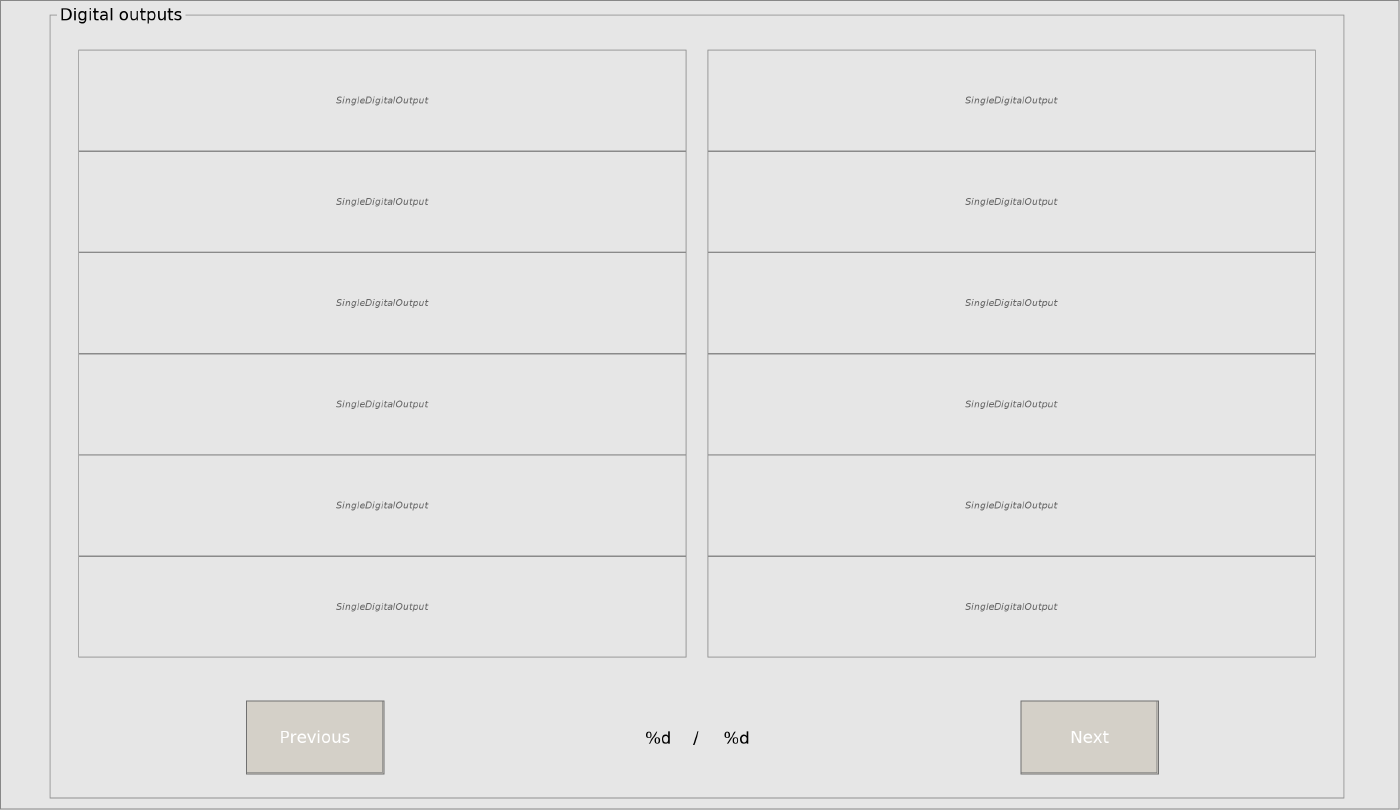
VISUALIZATION PageManualOutputs  // 1520x880
VAR_IN_OUT
	btnPrevious			: BOOL;
	btnNext				: BOOL;
	
	bPreviousInvisible	: BOOL;
	bNextInvisible		: BOOL;
	
	stDigitalOutputEmpty: ARRAY[1..12] OF BOOL;
	stDigitalOutputData	: ARRAY[1..12] OF ST_VisuCtrlOutputFrame;
	
	iOutputSelectedPageIndex	: USINT;
	iOutputTotalPageIndex 		: USINT;
END_VAR
    GroupBox (54,8 1405x859), "Digital outputs"
        Rectangle (721,769 50x50), "%d", text variable: iOutputTotalPageIndex + 1
        Rectangle (636,769 50x50), "%d", text variable: iOutputSelectedPageIndex+1
        Rectangle (636,768 131x51), "/"
        Button (213,753 150x80), "Previous", invisible if: bPreviousInvisible
            tap btnPrevious
        Button (1054,753 150x80), "Next", invisible if: bNextInvisible
            tap btnNext
        Frame (31,46 660x110), invisible if: stDigitalOutputEmpty[1]
            shows SingleDigitalOutput(stDigitalOutput := stDigitalOutputData[1])
        Frame (31,156 660x110), invisible if: stDigitalOutputEmpty[2]
            shows SingleDigitalOutput(stDigitalOutput := stDigitalOutputData[2])
        Frame (31,266 660x110), invisible if: stDigitalOutputEmpty[3]
            shows SingleDigitalOutput(stDigitalOutput := stDigitalOutputData[3])
        Frame (31,376 660x110), invisible if: stDigitalOutputEmpty[4]
            shows SingleDigitalOutput(stDigitalOutput := stDigitalOutputData[4])
        Frame (31,486 660x110), invisible if: stDigitalOutputEmpty[5]
            shows SingleDigitalOutput(stDigitalOutput := stDigitalOutputData[5])
        Frame (31,596 660x110), invisible if: stDigitalOutputEmpty[6]
            shows SingleDigitalOutput(stDigitalOutput := stDigitalOutputData[6])
        Frame (714,46 660x110), invisible if: stDigitalOutputEmpty[7]
            shows SingleDigitalOutput(stDigitalOutput := stDigitalOutputData[7])
    Frame (768,164 660x110), invisible if: stDigitalOutputEmpty[8]
        shows SingleDigitalOutput(stDigitalOutput := stDigitalOutputData[8])
    Frame (768,274 660x110), invisible if: stDigitalOutputEmpty[9]
        shows SingleDigitalOutput(stDigitalOutput := stDigitalOutputData[9])
    Frame (768,384 660x110), invisible if: stDigitalOutputEmpty[10]
        shows SingleDigitalOutput(stDigitalOutput := stDigitalOutputData[10])
    Frame (768,494 660x110), invisible if: stDigitalOutputEmpty[11]
        shows SingleDigitalOutput(stDigitalOutput := stDigitalOutputData[11])
    Frame (768,604 660x110), invisible if: stDigitalOutputEmpty[12]
        shows SingleDigitalOutput(stDigitalOutput := stDigitalOutputData[12])
END_VISUALIZATION

(* stored: Version 1.1.0.1, ProductVersion 3.1.4024.9
   Visu PageManualOutputs: Id {0c65fc21-68d0-4bdf-afcc-2296298a9986} *)
